# EPICS alarm handler configuration: css_share/detectors/SVT/alh/SVT.R4.alhConfig
GROUP NULL R4
INCLUDE R4 SVT.R4.S1.alhConfig
INCLUDE R4 SVT.R4.S2.alhConfig
INCLUDE R4 SVT.R4.S3.alhConfig
INCLUDE R4 SVT.R4.S4.alhConfig
INCLUDE R4 SVT.R4.S5.alhConfig
INCLUDE R4 SVT.R4.S6.alhConfig
INCLUDE R4 SVT.R4.S7.alhConfig
INCLUDE R4 SVT.R4.S8.alhConfig
INCLUDE R4 SVT.R4.S9.alhConfig
INCLUDE R4 SVT.R4.S10.alhConfig
INCLUDE R4 SVT.R4.S11.alhConfig
INCLUDE R4 SVT.R4.S12.alhConfig
INCLUDE R4 SVT.R4.S13.alhConfig
INCLUDE R4 SVT.R4.S14.alhConfig
INCLUDE R4 SVT.R4.S15.alhConfig
INCLUDE R4 SVT.R4.S16.alhConfig
INCLUDE R4 SVT.R4.S17.alhConfig
INCLUDE R4 SVT.R4.S18.alhConfig
INCLUDE R4 SVT.R4.S19.alhConfig
INCLUDE R4 SVT.R4.S20.alhConfig
INCLUDE R4 SVT.R4.S21.alhConfig
INCLUDE R4 SVT.R4.S22.alhConfig
INCLUDE R4 SVT.R4.S23.alhConfig
INCLUDE R4 SVT.R4.S24.alhConfig
